TYPE RecipeAssignment :
STRUCT
	LineIndex : INT;
	Name : T_MaxString;
	Value : T_MaxString;
	TableRows : INT;
END_STRUCT
END_TYPE

(* stored: Version 1.1.0.1
   DUT RecipeAssignment: Id {b038c5b2-303d-0e0f-36ad-357219138270} *)
